PROGRAM WAIT
VAR
	TON1: TON;
	WAIT_ENABLE: BOOL;
	
	count: INT;
END_VAR


TON1(IN:= TRUE , PT:=T#1MS , Q=> , ET=> );
IF TON1.Q THEN
	TON1(in:= FALSE);
	count := count + 1;
END_IF
//count := count + 1;

END_PROGRAM

(* stored: Version 1.1.0.1, ProductVersion 3.1.4024.0
   POU WAIT: Id {1ccdcde2-6e0b-48d8-a4a4-5efac2b2af7d}, SpecialFunc None *)
